// TIA Portal V20 export
FUNCTION_BLOCK "LER_SimActuator"   // FB114, LAD
// stored: Access Published, MemoryReserve 100, SetENOAutomatically false
   VAR_INPUT
      cmdHomePos : Bool;
      cmdWorkPos : Bool;
   END_VAR
   VAR_OUTPUT
      homePos : Bool;
      WorkPos : Bool;
   END_VAR
   VAR
      instTON { S7_SetPoint := 'True'} : Array[0..9] of TON_TIME;
      bitt { S7_SetPoint := 'True'} : Array[0..1] of Bool;
   END_VAR
   VAR CONSTANT
      delayTime : Time := T#20ms;
   END_VAR
   VAR_TEMP   // added for the SCL form of the ladder/FBD networks
      _w1 : Bool;
      _w2 : Bool;
   END_VAR
BEGIN

REGION Network 1: Sylinder
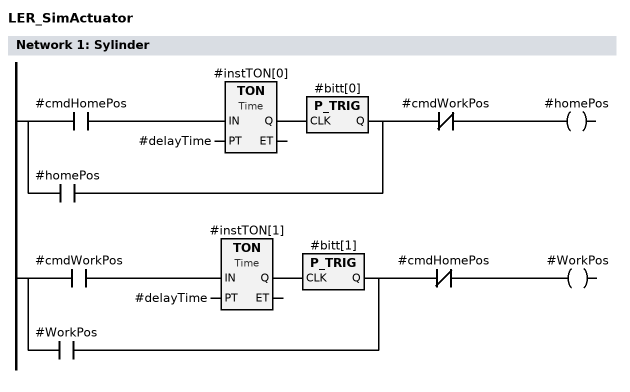
   RUNG wire#powerrail
      Contact( #cmdHomePos )
      { S7_Templates := "time_type := Time" } #instTON[0].TON(pt := #delayTime, et =>)
      P_Trig( #bitt[0] )
      wire#w1
      I_Contact( #cmdWorkPos )
      Coil( #homePos )
   END_RUNG
   RUNG wire#powerrail
      Contact( #homePos )
   END_RUNG wire#w1
   RUNG wire#powerrail
      Contact( #cmdWorkPos )
      { S7_Templates := "time_type := Time" } #instTON[1].TON(pt := #delayTime, et =>)
      P_Trig( #bitt[1] )
      wire#w2
      I_Contact( #cmdHomePos )
      Coil( #WorkPos )
   END_RUNG
   RUNG wire#powerrail
      Contact( #WorkPos )
   END_RUNG wire#w2
   // the same network as SCL:
   #instTON[0].TON(IN := #cmdHomePos, PT := #delayTime);
   #_w1 := #instTON[0].Q AND NOT #bitt[0];   // rising edge
   #bitt[0] := #instTON[0].Q;
   #homePos := (#_w1 OR #homePos) AND NOT #cmdWorkPos;
   #instTON[1].TON(IN := #cmdWorkPos, PT := #delayTime);
   #_w2 := #instTON[1].Q AND NOT #bitt[1];   // rising edge
   #bitt[1] := #instTON[1].Q;
   #WorkPos := (#_w2 OR #WorkPos) AND NOT #cmdHomePos;
END_REGION
END_FUNCTION_BLOCK
